FUNCTION AGILOG_DebugStart : BOOL
VAR_INPUT
	i_fileName :STRING;
END_VAR

IF GVL_RunTimeLogger.g_enableDebugLog THEN
	RETURN;
END_IF

GVL_RunTimeLogger.g_debugLogFileName  := i_fileName;

GVL_RunTimeLogger.g_debugLogReady := FALSE;
GVL_RunTimeLogger.g_debugLogBufferLock  :=FALSE;
GVL_RunTimeLogger.g_debugLogBufferInPtr :=1;
GVL_RunTimeLogger.g_debugLogBufferOutPtr :=1;


GVL_RunTimeLogger.g_enableDebugLog := TRUE;

END_FUNCTION

(* stored: Version 1.1.0.1, ProductVersion 3.1.4024.12
   POU AGILOG_DebugStart: Id {8ea148c4-efe5-435b-958b-9929af76f822}, SpecialFunc None *)
